// Mitsubishi GX Works2 project: IHW2   PLC: Q03UDE

// global labels: Global1
VAR_GLOBAL
  START AT X50 : BOOL;
  ESTOP AT X51 : BOOL;
  CB_A AT X52 : BOOL;
  CB_B AT X53 : BOOL;
  CB_C AT X54 : BOOL;
  CB_D AT X55 : BOOL;
  XX AT Y40 : BOOL;
  LL AT Y41 : BOOL;
  PP AT Y42 : BOOL;
  TT AT Y43 : BOOL;
  STOPBUT AT X56 : BOOL;
END_VAR

PROGRAM MAIN
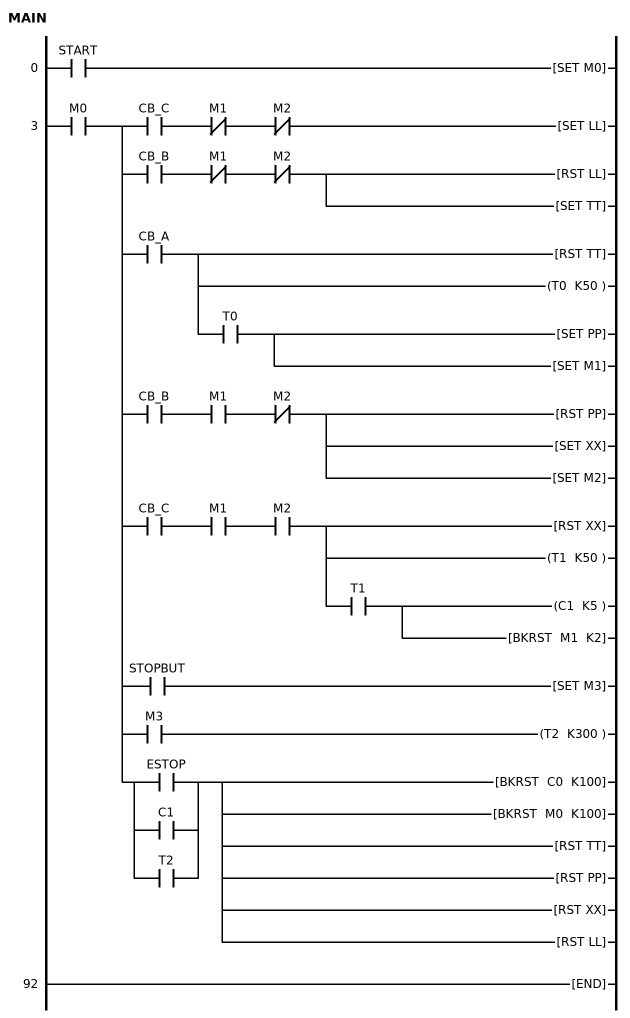
0     LD      START
      SET     M0
3     LD      M0
      MPS
      AND     CB_C
      ANI     M1
      ANI     M2
      SET     LL
      MRD
      AND     CB_B
      ANI     M1
      ANI     M2
      RST     LL
      SET     TT
      MRD
      AND     CB_A
      RST     TT
      OUT     T0 K50
      AND     T0
      SET     PP
      SET     M1
      MRD
      AND     CB_B
      AND     M1
      ANI     M2
      RST     PP
      SET     XX
      SET     M2
      MRD
      AND     CB_C
      AND     M1
      AND     M2
      RST     XX
      OUT     T1 K50
      AND     T1
      OUT     C1 K5
      BKRST   M1 K2
      MRD
      AND     STOPBUT
      SET     M3
      MRD
      AND     M3
      OUT     T2 K300
      MPP
      LD      ESTOP
      OR      C1
      OR      T2
      ANB
      BKRST   C0 K100
      BKRST   M0 K100
      RST     TT
      RST     PP
      RST     XX
      RST     LL
92    END
END_PROGRAM
